(* CODESYS project Untitled1.project

Project tree, tasks and I/O mapping:
  Device : CODESYS Control Win V3, 3S - Smart Software Solutions GmbH, order no. 305021, version 3.5.11.30
    application Application
      libraries: Standard, * (System)
      task MainTask (cyclic, interval t#20ms, priority 1) calls PLC_PRG
      program PLC_PRG [ST]
      global variables VarGlobais
      function block MyBlk [ST]
*)

// Device/Application/VarGlobais
{attribute 'qualified_only'}
VAR_GLOBAL
	VAR1 : REAL := 10.0;
	
END_VAR

VAR_GLOBAL CONSTANT
	CONST1 : REAL := 20.0;
END_VAR

// Device/Application/PLC_PRG
PROGRAM PLC_PRG
VAR
	VAR2 : REAL;
	T1 : MyBlk;
	PERIODO: TIME := T#10S;
	B1: BOOL ;
	R1: R_TRIG;
	T1Q : BOOL;
	ET1 : TIME;
	
END_VAR

VAR2 := VarGlobais.VAR1 + 10;

T1(IN := B1, PT:=PERIODO, Q => T1Q, ET => ET1);

R1(CLK:=T1.Q);

END_PROGRAM

// Device/Application/MyBlk
FUNCTION_BLOCK MyBlk
VAR_INPUT
	IN: BOOL;
	PT:TIME;
END_VAR
VAR_OUTPUT
	Q: BOOL;
	ET: TIME;
END_VAR
VAR
END_VAR

END_FUNCTION_BLOCK
